PROGRAM MAIN
VAR
END_VAR

END_PROGRAM

(* stored: Version 1.1.0.1
   POU MAIN: Id {4407b867-cc15-460f-9252-be64e4b0549b} *)
